// Struckig
// Copyright (C) 2022 Stefan Besler

// This program is free software: you can redistribute it and/or modify
// it under the terms of the GNU General Public License as published by
// the Free Software Foundation, either version 3 of the License, or
// (at your option) any later version.

// This program is distributed in the hope that it will be useful,
// but WITHOUT ANY WARRANTY; without even the implied warranty of
// MERCHANTABILITY or FITNESS FOR A PARTICULAR PURPOSE.  See the
// GNU General Public License for more details.
//
// You should have received a copy of the GNU General Public License
// along with THIS PROGRAM.  IF NOT, see <http://www.gnu.org/licenses/>.
{attribute 'qualified_only'}
{attribute 'strict'}
/// Defines the controlled state variables for trajectory generation.
/// The selected mode changes which boundary values and limits are interpreted
/// during validation and profile generation.
TYPE ControlInterfaceType :
(
  Undefined, //< Use global/default configuration.
  Position, //< Full control over position, velocity, and acceleration.
  Velocity //< Controls only velocity and acceleration states.
);
END_TYPE

(* stored: Version 1.1.0.1
   DUT ControlInterfaceType: Id {fa41777e-c926-434f-898a-1e6e98888ce1} *)
